Universal Robots PolyScope program: ad_tcp_62.urp

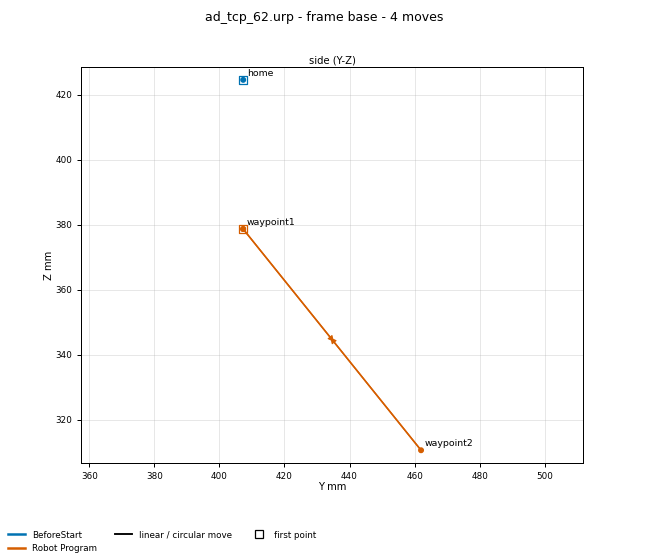
[picture p0: tool path of ad_tcp_62.urp in frame base, 4 of 4 moves have a stored position in this frame; points joined in program order, loops and branches not executed]
Program ad_tcp_62 (createdIn=3.2.19293 lastSavedIn=3.2.19293 directory=/programs installation=default robotSerialNumber=2015351391)
Calibrated DH parameters: a=[0.000352, -0.161198, -0.373486, 0.00005, 0.000049, 0]; d=[0.089268, 352.477598, -320.08558, -32.281492, 0.094939, 0.082518]; alpha=[1.570728, 0.001116, -0.003686, 1.571189, -1.570572, 0]; deltaTheta=[-0.000012, 1.181849, -1.491165, 0.309495, -0.000007, 0.000025]
BeforeStart
  tcp := 1
  tcp1 := p[0.15,0,0.15,0,0,0]
  tcp2 := p[-0.2,0,0.14,0,d2r(-25),0]
  MoveJ speed 60 deg/s, acceleration 80 deg/s^2 (recalculateMotions=false)
    Waypoint home: TCP in base x=-34.55 y=407.322 z=424.548 mm, rx=-2.361 ry=-1.6283 rz=0.0533 rad; joints [107.176, -73.328, -91.187, -91.149, 96.37, -51.236] deg; flange x=-11.66 y=382.141 z=544.853 mm, rx=-2.3609 ry=-1.6283 rz=0.0531 rad
Robot Program (runOnlyOnce=false motionType=MoveJ speed=1.047198 acceleration=1.396263 recalculateMotions=false)
  If tcp≟1
    Script: set_tcp(tcp1)
    tcp := 2
  ElseIf tcp≟2
    Script: set_tcp(tcp2)
    tcp := 1
  MoveL speed 250 mm/s, acceleration 1200 mm/s^2 (recalculateMotions=false) feature=Base
    Waypoint waypoint1: TCP in base x=-34.54 y=407.306 z=378.689 mm, rx=-2.3609 ry=-1.6283 rz=0.0532 rad; joints [107.173, -72.015, -98.934, -84.719, 96.378, -51.26] deg; flange x=-11.66 y=382.141 z=498.957 mm, rx=-2.3609 ry=-1.6283 rz=0.0531 rad
    Waypoint waypoint2: TCP in base x=-34.552 y=461.991 z=310.685 mm, rx=-2.361 ry=-1.6284 rz=0.0533 rad; joints [104.883, -79.338, -103.478, -73.127, 96.965, -53.542] deg; flange x=-11.66 y=436.853 z=431.022 mm, rx=-2.3609 ry=-1.6283 rz=0.0531 rad
    Waypoint waypoint1: TCP in base x=-34.54 y=407.306 z=378.689 mm, rx=-2.3609 ry=-1.6283 rz=0.0532 rad; joints [107.173, -72.015, -98.934, -84.719, 96.378, -51.26] deg; flange x=-11.66 y=382.141 z=498.957 mm, rx=-2.3609 ry=-1.6283 rz=0.0531 rad
